PROGRAM MAIN
VAR
	Data :fbData;
END_VAR

Data();

END_PROGRAM

(* stored: Version 1.1.0.1, ProductVersion 3.1.4024.6
   POU MAIN: Id {70a7c993-437c-4ccb-8a12-e68d1ba9b2d5}, SpecialFunc None *)
